// TIA Portal V21 export
VAR_GLOBAL   // PLC tag table "KAllGenZona"
END_VAR
VAR_GLOBAL CONSTANT   // user constants
   KALLGenZona_Prelavorazione_01 : Int := 1;   // Hello / Ciao
END_VAR
